// TIA Portal V20 export
// export: Created 2025-12-01T14:57:11.0834695Z, ExportSetting None, DisplayName Totally Integrated Automation Portal, DisplayVersion V20 Update 3, DisplayName TIA Portal Openness, DisplayVersion V20 Update 3, DisplayName TIA Portal Version Control Interface, DisplayVersion V20 Update 3, DisplayName STEP 7 Professional, DisplayVersion V20 Update 3, DisplayName STEP 7 Safety, DisplayVersion V20 Update 2, DisplayName WinCC Basic/Comfort/Advanced, DisplayVersion V20 Update 3, DisplayName WinCC Professional, DisplayVersion V20 Update 3, DisplayName WinCC Unified, DisplayVersion V20 Update 3
FUNCTION "FC725_CambiarUT_DePosicion" : Void   // FC725, LAD
TITLE = "CambiarUT_DePoscion"
{ S7_Optimized_Access := 'FALSE' }
AUTHOR : TRACKING
NAME : 20130301
VERSION : 3.0
// stored: AutoNumber false, SetENOAutomatically false
   VAR_INPUT
      NumeroUT : UInt;   // Numero de UT
      Posicion : UInt;   // Nueva Posicion
   END_VAR
   VAR_TEMP
      PosUT_Actual : UInt;
      Mesa : UInt;
      UT_Anterior : UInt;
      UT_Siguiente : UInt;
      NumeroTMP : UInt;
   END_VAR
BEGIN

NETWORK
TITLE = Inicializar
////////////////////////////////////////////////////////////////////////
////////////////////////////////////////////////////////////////////////
////////////////////////////////////////////////////////////////////////
// Inicilizar los numeros de DB's



NETWORK
TITLE = Sacar la UT de la Mesa Antigua
////////////////////////////////////////////////////////////////////////
////////////////////////////////////////////////////////////////////////
////////////////////////////////////////////////////////////////////////
// Sacar de la Mesa Antigua
      L     "DB812_UTs_Control".UT[#NumeroUT].MesaActual;
      L     "CTE_OffsetMesa";
      -I;
      T     #Mesa;

      L     "DB812_UTs_Control".UT[#NumeroUT].UT_AnteriorMesa;
      T     #UT_Anterior;
      L     "DB812_UTs_Control".UT[#NumeroUT].UT_SiguienteMesa;
      T     #UT_Siguiente;

      L     0;  // Inicializo
      T     "DB812_UTs_Control".UT[#NumeroUT].UT_AnteriorMesa;
      T     "DB812_UTs_Control".UT[#NumeroUT].UT_SiguienteMesa;




NETWORK
TITLE = --- Modificar Datos de la UT Anterior
////////////////////////////////////////////////////////////////////////
////////////////////////////////////////////////////////////////////////
////////////////////////////////////////////////////////////////////////
// Modificar Datos de la UT Anterior

      L     #UT_Anterior;
      L     0;  // Primera de la mesa
      <>I;
      JC    NoPrimeraUT_AnteriorUT_EnColaMesaOrigen;
      JU    PrimeraUT_AnteriorUT_EnColaMesaOrigen;


////////////////////////////////////////////////////////////////////////
// No existe ninguna UT Anterior en la Mesa Origen : Era la Primera
PrimeraUT_AnteriorUT_EnColaMesaOrigen:NOP   0;
      L     #UT_Siguiente;
      T     "DB810_ColasMesas".Colas[#Mesa].UT_PrimeraMesa;

      JU    Final_AnteriorUT_EnColaMesaOrigen;


////////////////////////////////////////////////////////////////////////
// Si existe UT Anterior en la Mesa Origen: No Era la Primera
NoPrimeraUT_AnteriorUT_EnColaMesaOrigen:NOP   0;
      L     #UT_Siguiente;
      T     "DB812_UTs_Control".UT[#UT_Anterior].UT_SiguienteMesa;

      JU    Final_AnteriorUT_EnColaMesaOrigen;


////////////////////////////////////////////////////////////////////////
// Final de la Modificacion de la Anterior UT
Final_AnteriorUT_EnColaMesaOrigen:NOP   0;



NETWORK
TITLE = --- Modificar Datos de la UT Siguiente
////////////////////////////////////////////////////////////////////////
////////////////////////////////////////////////////////////////////////
////////////////////////////////////////////////////////////////////////
// Modificar Datos de la UT Siguiente

      L     #UT_Siguiente;
      L     0;  // Es la ultima de la mesa
      ==I;
      JC    UltimaUT_SiguienteUT_EnColaMesaOrigen;
      JU    NoUltimaUT_SiguienteUT_EnColaMesaOrigen;


////////////////////////////////////////////////////////////////////////
// Si existe UT Siguiente en la Mesa Origen: No es la Ultima
UltimaUT_SiguienteUT_EnColaMesaOrigen:NOP   0;
      JU    Final_SiguienteUT_EnColaMesaOrigen;


////////////////////////////////////////////////////////////////////////
// Si existe UT Siguiente en la Mesa Origen: No es la Ultima
NoUltimaUT_SiguienteUT_EnColaMesaOrigen:NOP   0;
      L     #UT_Anterior;
      T     "DB812_UTs_Control".UT[#UT_Siguiente].UT_AnteriorMesa;

      JU    Final_SiguienteUT_EnColaMesaOrigen;


////////////////////////////////////////////////////////////////////////
// Final de la Modificacion de la Anterior UT
Final_SiguienteUT_EnColaMesaOrigen:NOP   0;




NETWORK
TITLE = Insertar en la Nueva Posicion --- Buscar la Nueva posicion
////////////////////////////////////////////////////////////////////////
////////////////////////////////////////////////////////////////////////
////////////////////////////////////////////////////////////////////////
// --- Buscar la Posicion
      L     "DB810_ColasMesas".Colas[#Mesa].UT_PrimeraMesa;
      T     #NumeroTMP;

      L     1;  // Inicializar Posicion
      T     #PosUT_Actual;


////////////////////////////////////////////////////////////////////////
// Bucle de Busqueda de Posicion para INSERTAR la UT
BucleBusquedaDePosicion_EnColaMesaDestino:NOP   0;
      L     #PosUT_Actual;
      L     #Posicion;
      ==I;  // Encontrada la Posicion
      JC    EncontradaPosicion_EnColaMesaDestino;

      L     "DB812_UTs_Control".UT[#NumeroTMP].UT_SiguienteMesa;
      L     0;
      ==I;  // Hay que Insertar en la Ultima Posicion ?
      JC    EnPosicionUltima_EnColaMesaDestino;

      L     "DB812_UTs_Control".UT[#NumeroTMP].UT_SiguienteMesa;
      T     #NumeroTMP;

      L     #PosUT_Actual;  // Incrementar la Posicion
      L     1;
      +I;
      T     #PosUT_Actual;

      JU    BucleBusquedaDePosicion_EnColaMesaDestino;



NETWORK
TITLE = --- Encontrada la Posicion
////////////////////////////////////////////////////////////////////////
////////////////////////////////////////////////////////////////////////
////////////////////////////////////////////////////////////////////////
// --- Posicion Encontrada
// --- Mirar en que Posicion esta (Primera, Intermedia, Ultima)

EncontradaPosicion_EnColaMesaDestino:NOP   0;
      L     "DB812_UTs_Control".UT[#NumeroTMP].UT_AnteriorMesa;
      L     0;
      ==I;  // Es la Primera Posicion ?
      JC    EnPosicionPrimera_EnColaMesaDestino;

// Es Posicion Intermedia
      JU    EnPosicionIntermedia_EnColaMesaDestino;



NETWORK
TITLE = --- En la Primera Posicion
EnPosicionPrimera_EnColaMesaDestino:NOP   0;

////////////////////////////////////////////////////////////////////////
////////////////////////////////////////////////////////////////////////
////////////////////////////////////////////////////////////////////////
// --- Insertar la UT en la Primera Posicion
// ---------- Modificar la Primera de la Mesa
// ---------- Modificar la UT que Estaba Primera
// ---------- Modificar la UT a insertar


////////////////////////////////////////////////////////////////////////
// ---------- Modificar la Primera de la Cola de la Mesa
      L     #NumeroUT;  // Es la primera de la Mesa
      T     "DB810_ColasMesas".Colas[#Mesa].UT_PrimeraMesa;

////////////////////////////////////////////////////////////////////////
// ---------- Modificar la UT que Estaba Primera
      L     #NumeroUT;
      T     "DB812_UTs_Control".UT[#NumeroTMP].UT_AnteriorMesa;

////////////////////////////////////////////////////////////////////////
// ---------- Modificar la UT a insertar
      L     0;
      T     "DB812_UTs_Control".UT[#NumeroUT].UT_AnteriorMesa;
      L     #NumeroTMP;
      T     "DB812_UTs_Control".UT[#NumeroUT].UT_SiguienteMesa;

////////////////////////////////////////////////////////////////////////
// ---------- Finalizado la Insercion de la UT
      JU    Final_Funcion;



NETWORK
TITLE = --- En la Ultima Posicion
EnPosicionUltima_EnColaMesaDestino:NOP   0;

////////////////////////////////////////////////////////////////////////
////////////////////////////////////////////////////////////////////////
////////////////////////////////////////////////////////////////////////
// --- Insertar la UT en la Ultima Posicion
// ---------- Modificar la Ultima UT de la Mesa
// ---------- Modificar la UT a insertar


////////////////////////////////////////////////////////////////////////
// ---------- Modificar la Ultima UT de la Mesa
      L     #NumeroUT;  // Aviso del que estaba primero
      T     "DB812_UTs_Control".UT[#NumeroTMP].UT_SiguienteMesa;

////////////////////////////////////////////////////////////////////////
// ---------- Modificar la UT a insertar
      L     #NumeroTMP;
      T     "DB812_UTs_Control".UT[#NumeroUT].UT_AnteriorMesa;
      L     0;
      T     "DB812_UTs_Control".UT[#NumeroUT].UT_SiguienteMesa;

////////////////////////////////////////////////////////////////////////
// ---------- Finalizado la Insercion de la UT
      JU    Final_Funcion;



NETWORK
TITLE = --- En la Posicion Intermedia
EnPosicionIntermedia_EnColaMesaDestino:NOP   0;

////////////////////////////////////////////////////////////////////////
////////////////////////////////////////////////////////////////////////
////////////////////////////////////////////////////////////////////////
// --- Insertar la UT en la Ultima Intermedia
// ---------- Recoger los Numeros De UT Anterior y Siguiente
// ---------- Modificar la UT Anterior que estaba en la Cola
// ---------- Modificar la UT Siguinete que estaba en la Cola
// ---------- Modificar la UT a Insertar


////////////////////////////////////////////////////////////////////////
// ---------- Recoger los Numeros De UT Anterior y Siguiente
      L     "DB812_UTs_Control".UT[#NumeroTMP].UT_AnteriorMesa;
      T     #UT_Anterior;
      L     "DB812_UTs_Control".UT[#NumeroTMP].UT_SiguienteMesa;
      T     #UT_Siguiente;

////////////////////////////////////////////////////////////////////////
// ---------- Modificar la UT Anterior que estaba en la Cola
      L     #NumeroUT;
      T     "DB812_UTs_Control".UT[#UT_Anterior].UT_SiguienteMesa;

////////////////////////////////////////////////////////////////////////
// ---------- Modificar la UT que se desplaza que estaba en la Cola
      L     #NumeroUT;
      T     "DB812_UTs_Control".UT[#NumeroTMP].UT_AnteriorMesa;

////////////////////////////////////////////////////////////////////////
// ---------- Modificar la UT a insertar
      L     #UT_Anterior;
      T     "DB812_UTs_Control".UT[#NumeroUT].UT_AnteriorMesa;
      L     #NumeroTMP;
      T     "DB812_UTs_Control".UT[#NumeroUT].UT_SiguienteMesa;

////////////////////////////////////////////////////////////////////////
// ---------- Finalizado la Insercion de la UT
      JU    Final_Funcion;



NETWORK
TITLE = Final de la funcion
////////////////////////////////////////////////////////////////////////
////////////////////////////////////////////////////////////////////////
////////////////////////////////////////////////////////////////////////
Final_Funcion:NOP   0;

END_FUNCTION
